// TIA Portal V20 export
// export: Created 2026-04-28T10:07:59.5032164Z, ExportSetting WithDefaults, DisplayName Totally Integrated Automation Portal, DisplayVersion V20, DisplayName TIA Portal Openness, DisplayVersion V20, DisplayName TIA Portal Version Control Interface, DisplayVersion V20, DisplayName SINAMICS Startdrive Advanced, DisplayVersion V20, DisplayName SINAMICS Startdrive G130, G150, S120, S150, SINAMICS MV, G220, S200, S210, DisplayVersion V20, DisplayName SINAMICS Startdrive G110M, G120, G120C, G120D, G120P, G115D, DisplayVersion V20, DisplayName STEP 7 Professional, DisplayVersion V20, DisplayName STEP 7 Safety, DisplayVersion V20, DisplayName WinCC Basic/Comfort/Advanced, DisplayVersion V20, DisplayName WinCC Unified, DisplayVersion V20
TYPE "Daten_SPT_10"
// stored: IsFailsafeCompliant false
   STRUCT
      xBurn : Bool;   // Selection Burner
      xHoAiTe : Bool;   // Selection Hot air temperature
      txt_rAlHoAi : DInt;   // Alarm Hot air
      txt_max_rAlHoAi : DInt;   // max. Alarm Hot air
      txt_min_rAlHoAi : DInt;   // min. Alarm Hot air
      xHotAirSoll : Bool;   // Select/ Hot air Set Value
      xHotAirIst : Bool;   // Select/ Hot air Actual Value
      txt_rHotAirSoll : DInt;   // Set Value Hot air
      txt_rHotAirSt1 : DInt;   // Set Value Hot air level 1
      txt_rHotAirSt2 : DInt;   // Set Value Hot air level 2
      txt_rHotAirSt3 : DInt;   // Set Value Hot air level 3
      txt_rHotAirSt4 : DInt;   // Set Value Hot air level 4
      RangeHotAir : DInt;   // Range Hot air
      xDeliFan : Bool;   // Selection Deli.Fan
      xDeliFanSoll : Bool;   // Selection Deli.Fan Set Value
      xDeliFanIst : Bool;   // Selection Deli.Fan Actual Value
      txt_rDeliFan : DInt;   // Set Value Deli.Fan
      RangeDeliFan : DInt;   // Range Deli.Fan
      xDiPrFiBu : Bool;   // Selection Differential pressure filter heating
      txt_rDiPrFiBu : DInt;   // Set Value Differential pressure filter heating
      txt_max_rDiPrFiBu : DInt;   // Differential pressure filter heating Input Limit
      RangeDiPrFiBu : DInt;   // Range Differential pressure filter heating
      xFlRaAirBurn : Bool;   // Selection Volume flow at the Heating
      RangeFlRaAirBurn : DInt;   // Range Volume flow at the Heating
      xTempBurn : Bool;   // Selection Inlet Temperatur Heating
      RangeTempBurn : DInt;   // Range Inlet Temperatur Heating
      xOptionTZ : Bool;   // Dorst Option
      iTakt_FlRaAirBurn : DInt;   // Interval for recording the measured values
      iAnzWerte_FlRaAirBurn : DInt;   // Number of measured values
      iTakt_TempBurn : DInt;   // Interval for recording the measured values
      iAnzWerte_TempBurn : DInt;   // Number of measured values
      iTakt_DeliFan : DInt;   // Interval for recording the measured values
      iAnzWerte_DeliFan : DInt;   // Number of measured values
      iTakt_HoAiTe : DInt;   // Interval for recording the measured values
      iAnzWerte_HoAiTe : DInt;   // Number of measured values
      iTakt_DiFiBurn : DInt;   // Interval for recording the measured values
      iAnzWerte_DiFiBurn : DInt;   // Number of measured values
      xGasRate : Bool;   // Selection Display total gas quantity
      RangeGasRate : Real;   // Range Display total gas quantity
      rGasRate_1 : Real;   // Display total gas quantity
      rGasRate_2 : Real;   // Display total gas quantity 2
      xTempRegSoft : Bool;   // Selection with software temperature controller
      rXp_Het : Real;   // Control P-Value Hot air controller
      rTi_Het : Real;   // Control I-Value Hot air controller
      rTd2_Het : Real;   // Control D-Value Hot air controller
      rRunStellMot : Real;   // Actuator running time
      xTempBurn_PT100 : Bool;   // Selection Temperatur Sensor with PT100
      cTempRegSoft : Int;   // Selection 0=hardware controller / 1=hot air / 2=residual humidity / 3=exhaust air
      rXP_HotAir : Real;   // Control P-Value Hot air controller
      rTi_HotAir : Real;   // Control I-Value Hot air controller
      rTd2_HotAir : Real;   // Control D-Value Hot air controller
      rXP_ReGrHu : Real;   // Control P-Value Hot air controller residual humidity
      rTi_ReGrHu : Real;   // Control I-Value Hot air controller residual humidity
      rTd2_ReGrHu : Real;   // Control D-Value Hot air controller residual humidity
      rXP_ExAir : Real;   // Control P-Value Hot air controller Exhaust air
      rTi_ExAir : Real;   // Control I-Value Hot air controller Exhaust air
      rTd2_ExAir : Real;   // Control D-Value Hot air controller Exhaust air
      xHardwareRegler : Bool;   // Hot air Controller 0=Software, 1=Hardware
      xCombAirFan : Bool;   // Option Verbrennungsluft Geblaese
      x_HoAiTeTB45 : Bool;   // Hot air monitoring TB45 Active 0=No, 1=Yes
      xBuCtrlExt : Bool;   // External start/stop button active 0=No, 1=Yes
      xDiPrFiBu_Sensor2 : Bool;   // Option: Selection of vacuum sensor type 2 -100 to 100 mBar Sensor type 2 = 1
      xEH_Option : Bool;   // Option: Select electric heating option 0=No, 1=Yes
      x_HoAiTeEHTB45 : Bool;   // Hot air monitoring electric heater TB45 Active 0=No, 1=Yes
      xMinHotAirTempMainOff : Bool;   // Option :Hot air temperature Min. for main fan off
      txt_rAlHoAi_D20 : DInt;   // Alarm Hot air
      txt_max_rAlHoAi_D20 : DInt;   // max. Alarm Hot air
      RangeHotAir_D20 : DInt;   // Range Hot air
      RangeGasRate_D20 : Real;   // Range Display total gas quantity
   END_STRUCT;
END_TYPE
